  583 = 'S2 583 Row 59 Lost Return Position... Check Ixxx.x Default' | German: 'S2 583 Row 59 Lost Return Position... Check Ixxx.x German' | French: 'S2 583 Row 59 Lost Return Position... Check Ixxx.x French'
  584 = 'S2 584 Row 59 Switch Fault... Check Ixxx.x / Ixxx.x Default' | German: 'S2 584 Row 59 Switch Fault... Check Ixxx.x / Ixxx.x German' | French: 'S2 584 Row 59 Switch Fault... Check Ixxx.x / Ixxx.x French'
  585 = 'S2 585 Row 59 Spare Message Default' | German: 'S2 585 Row 59 Spare Message German' | French: 'S2 585 Row 59 Spare Message French'
  586 = 'S2 586 Row 59 Spare Message Default' | German: 'S2 586 Row 59 Spare Message German' | French: 'S2 586 Row 59 Spare Message French'
  587 = 'S2 587 Row 59 Spare Message Default' | German: 'S2 587 Row 59 Spare Message German' | French: 'S2 587 Row 59 Spare Message French'
  588 = 'S2 588 Row 59 Spare Message Default' | German: 'S2 588 Row 59 Spare Message German' | French: 'S2 588 Row 59 Spare Message French'
  589 = 'S2 589 Row 59 Spare Message Default' | German: 'S2 589 Row 59 Spare Message German' | French: 'S2 589 Row 59 Spare Message French'
  590 = 'S2 590 Row 60 Failed To Advance.. Check Qxxx.x Default' | German: 'S2 590 Row 60 Failed To Advance.. Check Qxxx.x German' | French: 'S2 590 Row 60 Failed To Advance.. Check Qxxx.x French'
  591 = 'S2 591 Row 60 Failed To Return.. Check Qxxx.x Default' | German: 'S2 591 Row 60 Failed To Return.. Check Qxxx.x German' | French: 'S2 591 Row 60 Failed To Return.. Check Qxxx.x French'
  592 = 'S2 592 Row 60 Lost Advance Position... Check Ixxx.x Default' | German: 'S2 592 Row 60 Lost Advance Position... Check Ixxx.x German' | French: 'S2 592 Row 60 Lost Advance Position... Check Ixxx.x French'
  593 = 'S2 593 Row 60 Lost Return Position... Check Ixxx.x Default' | German: 'S2 593 Row 60 Lost Return Position... Check Ixxx.x German' | French: 'S2 593 Row 60 Lost Return Position... Check Ixxx.x French'
  594 = 'S2 594 Row 60 Switch Fault... Check Ixxx.x / Ixxx.x Default' | German: 'S2 594 Row 60 Switch Fault... Check Ixxx.x / Ixxx.x German' | French: 'S2 594 Row 60 Switch Fault... Check Ixxx.x / Ixxx.x French'
  595 = 'S2 595 Row 60 Spare Message Default' | German: 'S2 595 Row 60 Spare Message German' | French: 'S2 595 Row 60 Spare Message French'
  596 = 'S2 596 Row 60 Spare Message Default' | German: 'S2 596 Row 60 Spare Message German' | French: 'S2 596 Row 60 Spare Message French'
  597 = 'S2 597 Row 60 Spare Message Default' | German: 'S2 597 Row 60 Spare Message German' | French: 'S2 597 Row 60 Spare Message French'
  598 = 'S2 598 Row 60 Spare Message Default' | German: 'S2 598 Row 60 Spare Message German' | French: 'S2 598 Row 60 Spare Message French'
  599 = 'S2 599 Row 60 Spare Message Default' | German: 'S2 599 Row 60 Spare Message German' | French: 'S2 599 Row 60 Spare Message French'
  600 = 'S2 600 Row 61 Failed To Advance.. Check Qxxx.x Default' | German: 'S2 600 Row 61 Failed To Advance.. Check Qxxx.x German' | French: 'S2 600 Row 61 Failed To Advance.. Check Qxxx.x French'
  601 = 'S2 601 Row 61 Failed To Return.. Check Qxxx.x Default' | German: 'S2 601 Row 61 Failed To Return.. Check Qxxx.x German' | French: 'S2 601 Row 61 Failed To Return.. Check Qxxx.x French'
  602 = 'S2 602 Row 61 Lost Advance Position... Check Ixxx.x Default' | German: 'S2 602 Row 61 Lost Advance Position... Check Ixxx.x German' | French: 'S2 602 Row 61 Lost Advance Position... Check Ixxx.x French'
  603 = 'S2 603 Row 61 Lost Return Position... Check Ixxx.x Default' | German: 'S2 603 Row 61 Lost Return Position... Check Ixxx.x German' | French: 'S2 603 Row 61 Lost Return Position... Check Ixxx.x French'
  604 = 'S2 604 Row 61 Switch Fault... Check Ixxx.x / Ixxx.x Default' | German: 'S2 604 Row 61 Switch Fault... Check Ixxx.x / Ixxx.x German' | French: 'S2 604 Row 61 Switch Fault... Check Ixxx.x / Ixxx.x French'
  605 = 'S2 605 Row 61 Spare Message Default' | German: 'S2 605 Row 61 Spare Message German' | French: 'S2 605 Row 61 Spare Message French'
  606 = 'S2 606 Row 61 Spare Message Default' | German: 'S2 606 Row 61 Spare Message German' | French: 'S2 606 Row 61 Spare Message French'
  607 = 'S2 607 Row 61 Spare Message Default' | German: 'S2 607 Row 61 Spare Message German' | French: 'S2 607 Row 61 Spare Message French'
  608 = 'S2 608 Row 61 Spare Message Default' | German: 'S2 608 Row 61 Spare Message German' | French: 'S2 608 Row 61 Spare Message French'
  609 = 'S2 609 Row 61 Spare Message Default' | German: 'S2 609 Row 61 Spare Message German' | French: 'S2 609 Row 61 Spare Message French'
  610 = 'S2 610 Row 62 Failed To Advance.. Check Qxxx.x Default' | German: 'S2 610 Row 62 Failed To Advance.. Check Qxxx.x German' | French: 'S2 610 Row 62 Failed To Advance.. Check Qxxx.x French'
  611 = 'S2 611 Row 62 Failed To Return.. Check Qxxx.x Default' | German: 'S2 611 Row 62 Failed To Return.. Check Qxxx.x German' | French: 'S2 611 Row 62 Failed To Return.. Check Qxxx.x French'
  612 = 'S2 612 Row 62 Lost Advance Position... Check Ixxx.x Default' | German: 'S2 612 Row 62 Lost Advance Position... Check Ixxx.x German' | French: 'S2 612 Row 62 Lost Advance Position... Check Ixxx.x French'
  613 = 'S2 613 Row 62 Lost Return Position... Check Ixxx.x Default' | German: 'S2 613 Row 62 Lost Return Position... Check Ixxx.x German' | French: 'S2 613 Row 62 Lost Return Position... Check Ixxx.x French'
  614 = 'S2 614 Row 62 Switch Fault... Check Ixxx.x / Ixxx.x Default' | German: 'S2 614 Row 62 Switch Fault... Check Ixxx.x / Ixxx.x German' | French: 'S2 614 Row 62 Switch Fault... Check Ixxx.x / Ixxx.x French'
  615 = 'S2 615 Row 62 Spare Message Default' | German: 'S2 615 Row 62 Spare Message German' | French: 'S2 615 Row 62 Spare Message French'
  616 = 'S2 616 Row 62 Spare Message Default' | German: 'S2 616 Row 62 Spare Message German' | French: 'S2 616 Row 62 Spare Message French'
  617 = 'S2 617 Row 62 Spare Message Default' | German: 'S2 617 Row 62 Spare Message German' | French: 'S2 617 Row 62 Spare Message French'
  618 = 'S2 618 Row 62 Spare Message Default' | German: 'S2 618 Row 62 Spare Message German' | French: 'S2 618 Row 62 Spare Message French'
  619 = 'S2 619 Row 62 Spare Message Default' | German: 'S2 619 Row 62 Spare Message German' | French: 'S2 619 Row 62 Spare Message French'
  620 = 'S2 620 Row 63 Failed To Advance.. Check Qxxx.x Default' | German: 'S2 620 Row 63 Failed To Advance.. Check Qxxx.x German' | French: 'S2 620 Row 63 Failed To Advance.. Check Qxxx.x French'
  621 = 'S2 621 Row 63 Failed To Return.. Check Qxxx.x Default' | German: 'S2 621 Row 63 Failed To Return.. Check Qxxx.x German' | French: 'S2 621 Row 63 Failed To Return.. Check Qxxx.x French'
  622 = 'S2 622 Row 63 Lost Advance Position... Check Ixxx.x Default' | German: 'S2 622 Row 63 Lost Advance Position... Check Ixxx.x German' | French: 'S2 622 Row 63 Lost Advance Position... Check Ixxx.x French'
  623 = 'S2 623 Row 63 Lost Return Position... Check Ixxx.x Default' | German: 'S2 623 Row 63 Lost Return Position... Check Ixxx.x German' | French: 'S2 623 Row 63 Lost Return Position... Check Ixxx.x French'
  624 = 'S2 624 Row 63 Switch Fault... Check Ixxx.x / Ixxx.x Default' | German: 'S2 624 Row 63 Switch Fault... Check Ixxx.x / Ixxx.x German' | French: 'S2 624 Row 63 Switch Fault... Check Ixxx.x / Ixxx.x French'
  625 = 'S2 625 Row 63 Spare Message Default' | German: 'S2 625 Row 63 Spare Message German' | French: 'S2 625 Row 63 Spare Message French'
  626 = 'S2 626 Row 63 Spare Message Default' | German: 'S2 626 Row 63 Spare Message German' | French: 'S2 626 Row 63 Spare Message French'
  627 = 'S2 627 Row 63 Spare Message Default' | German: 'S2 627 Row 63 Spare Message German' | French: 'S2 627 Row 63 Spare Message French'
  628 = 'S2 628 Row 63 Spare Message Default' | German: 'S2 628 Row 63 Spare Message German' | French: 'S2 628 Row 63 Spare Message French'
  629 = 'S2 629 Row 63 Spare Message Default' | German: 'S2 629 Row 63 Spare Message German' | French: 'S2 629 Row 63 Spare Message French'
  630 = 'S2 630 Row 64 Failed To Advance.. Check Qxxx.x Default' | German: 'S2 630 Row 64 Failed To Advance.. Check Qxxx.x German' | French: 'S2 630 Row 64 Failed To Advance.. Check Qxxx.x French'
  631 = 'S2 631 Row 64 Failed To Return.. Check Qxxx.x Default' | German: 'S2 631 Row 64 Failed To Return.. Check Qxxx.x German' | French: 'S2 631 Row 64 Failed To Return.. Check Qxxx.x French'
  632 = 'S2 632 Row 64 Lost Advance Position... Check Ixxx.x Default' | German: 'S2 632 Row 64 Lost Advance Position... Check Ixxx.x German' | French: 'S2 632 Row 64 Lost Advance Position... Check Ixxx.x French'
  633 = 'S2 633 Row 64 Lost Return Position... Check Ixxx.x Default' | German: 'S2 633 Row 64 Lost Return Position... Check Ixxx.x German' | French: 'S2 633 Row 64 Lost Return Position... Check Ixxx.x French'
  634 = 'S2 634 Row 64 Switch Fault... Check Ixxx.x / Ixxx.x Default' | German: 'S2 634 Row 64 Switch Fault... Check Ixxx.x / Ixxx.x German' | French: 'S2 634 Row 64 Switch Fault... Check Ixxx.x / Ixxx.x French'
  635 = 'S2 635 Row 64 Spare Message Default' | German: 'S2 635 Row 64 Spare Message German' | French: 'S2 635 Row 64 Spare Message French'
  636 = 'S2 636 Row 64 Spare Message Default' | German: 'S2 636 Row 64 Spare Message German' | French: 'S2 636 Row 64 Spare Message French'
  637 = 'S2 637 Row 64 Spare Message Default' | German: 'S2 637 Row 64 Spare Message German' | French: 'S2 637 Row 64 Spare Message French'
  638 = 'S2 638 Row 64 Spare Message Default' | German: 'S2 638 Row 64 Spare Message German' | French: 'S2 638 Row 64 Spare Message French'
  639 = 'S2 639 Row 64 Spare Message Default' | German: 'S2 639 Row 64 Spare Message German' | French: 'S2 639 Row 64 Spare Message French'
  640 = 'S2 640 Row 65 Failed To Advance.. Check Qxxx.x Default' | German: 'S2 640 Row 65 Failed To Advance.. Check Qxxx.x German' | French: 'S2 640 Row 65 Failed To Advance.. Check Qxxx.x French'
  641 = 'S2 641 Row 65 Failed To Return.. Check Qxxx.x Default' | German: 'S2 641 Row 65 Failed To Return.. Check Qxxx.x German' | French: 'S2 641 Row 65 Failed To Return.. Check Qxxx.x French'
  642 = 'S2 642 Row 65 Lost Advance Position... Check Ixxx.x Default' | German: 'S2 642 Row 65 Lost Advance Position... Check Ixxx.x German' | French: 'S2 642 Row 65 Lost Advance Position... Check Ixxx.x French'
  643 = 'S2 643 Row 65 Lost Return Position... Check Ixxx.x Default' | German: 'S2 643 Row 65 Lost Return Position... Check Ixxx.x German' | French: 'S2 643 Row 65 Lost Return Position... Check Ixxx.x French'
  644 = 'S2 644 Row 65 Switch Fault... Check Ixxx.x / Ixxx.x Default' | German: 'S2 644 Row 65 Switch Fault... Check Ixxx.x / Ixxx.x German' | French: 'S2 644 Row 65 Switch Fault... Check Ixxx.x / Ixxx.x French'
  645 = 'S2 645 Row 65 Spare Message Default' | German: 'S2 645 Row 65 Spare Message German' | French: 'S2 645 Row 65 Spare Message French'
  646 = 'S2 646 Row 65 Spare Message Default' | German: 'S2 646 Row 65 Spare Message German' | French: 'S2 646 Row 65 Spare Message French'
  647 = 'S2 647 Row 65 Spare Message Default' | German: 'S2 647 Row 65 Spare Message German' | French: 'S2 647 Row 65 Spare Message French'
  648 = 'S2 648 Row 65 Spare Message Default' | German: 'S2 648 Row 65 Spare Message German' | French: 'S2 648 Row 65 Spare Message French'
  649 = 'S2 649 Row 65 Spare Message Default' | German: 'S2 649 Row 65 Spare Message German' | French: 'S2 649 Row 65 Spare Message French'
  650 = 'S2 650 Row 66 Failed To Advance.. Check Qxxx.x Default' | German: 'S2 650 Row 66 Failed To Advance.. Check Qxxx.x German' | French: 'S2 650 Row 66 Failed To Advance.. Check Qxxx.x French'
  651 = 'S2 651 Row 66 Failed To Return.. Check Qxxx.x Default' | German: 'S2 651 Row 66 Failed To Return.. Check Qxxx.x German' | French: 'S2 651 Row 66 Failed To Return.. Check Qxxx.x French'
  652 = 'S2 652 Row 66 Lost Advance Position... Check Ixxx.x Default' | German: 'S2 652 Row 66 Lost Advance Position... Check Ixxx.x German' | French: 'S2 652 Row 66 Lost Advance Position... Check Ixxx.x French'
  653 = 'S2 653 Row 66 Lost Return Position... Check Ixxx.x Default' | German: 'S2 653 Row 66 Lost Return Position... Check Ixxx.x German' | French: 'S2 653 Row 66 Lost Return Position... Check Ixxx.x French'
  654 = 'S2 654 Row 66 Switch Fault... Check Ixxx.x / Ixxx.x Default' | German: 'S2 654 Row 66 Switch Fault... Check Ixxx.x / Ixxx.x German' | French: 'S2 654 Row 66 Switch Fault... Check Ixxx.x / Ixxx.x French'
  655 = 'S2 655 Row 66 Spare Message Default' | German: 'S2 655 Row 66 Spare Message German' | French: 'S2 655 Row 66 Spare Message French'
  656 = 'S2 656 Row 66 Spare Message Default' | German: 'S2 656 Row 66 Spare Message German' | French: 'S2 656 Row 66 Spare Message French'
  657 = 'S2 657 Row 66 Spare Message Default' | German: 'S2 657 Row 66 Spare Message German' | French: 'S2 657 Row 66 Spare Message French'
  658 = 'S2 658 Row 66 Spare Message Default' | German: 'S2 658 Row 66 Spare Message German' | French: 'S2 658 Row 66 Spare Message French'
  659 = 'S2 659 Row 66 Spare Message Default' | German: 'S2 659 Row 66 Spare Message German' | French: 'S2 659 Row 66 Spare Message French'
  660 = 'S2 660 Row 67 Failed To Advance.. Check Qxxx.x Default' | German: 'S2 660 Row 67 Failed To Advance.. Check Qxxx.x German' | French: 'S2 660 Row 67 Failed To Advance.. Check Qxxx.x French'
  661 = 'S2 661 Row 67 Failed To Return.. Check Qxxx.x Default' | German: 'S2 661 Row 67 Failed To Return.. Check Qxxx.x German' | French: 'S2 661 Row 67 Failed To Return.. Check Qxxx.x French'
  662 = 'S2 662 Row 67 Lost Advance Position... Check Ixxx.x Default' | German: 'S2 662 Row 67 Lost Advance Position... Check Ixxx.x German' | French: 'S2 662 Row 67 Lost Advance Position... Check Ixxx.x French'
  663 = 'S2 663 Row 67 Lost Return Position... Check Ixxx.x Default' | German: 'S2 663 Row 67 Lost Return Position... Check Ixxx.x German' | French: 'S2 663 Row 67 Lost Return Position... Check Ixxx.x French'
  664 = 'S2 664 Row 67 Switch Fault... Check Ixxx.x / Ixxx.x Default' | German: 'S2 664 Row 67 Switch Fault... Check Ixxx.x / Ixxx.x German' | French: 'S2 664 Row 67 Switch Fault... Check Ixxx.x / Ixxx.x French'
  665 = 'S2 665 Row 67 Spare Message Default' | German: 'S2 665 Row 67 Spare Message German' | French: 'S2 665 Row 67 Spare Message French'
  666 = 'S2 666 Row 67 Spare Message Default' | German: 'S2 666 Row 67 Spare Message German' | French: 'S2 666 Row 67 Spare Message French'
  667 = 'S2 667 Row 67 Spare Message Default' | German: 'S2 667 Row 67 Spare Message German' | French: 'S2 667 Row 67 Spare Message French'
  668 = 'S2 668 Row 67 Spare Message Default' | German: 'S2 668 Row 67 Spare Message German' | French: 'S2 668 Row 67 Spare Message French'
  669 = 'S2 669 Row 67 Spare Message Default' | German: 'S2 669 Row 67 Spare Message German' | French: 'S2 669 Row 67 Spare Message French'
  670 = 'S2 670 Row 68 Failed To Advance.. Check Qxxx.x Default' | German: 'S2 670 Row 68 Failed To Advance.. Check Qxxx.x German' | French: 'S2 670 Row 68 Failed To Advance.. Check Qxxx.x French'
  671 = 'S2 671 Row 68 Failed To Return.. Check Qxxx.x Default' | German: 'S2 671 Row 68 Failed To Return.. Check Qxxx.x German' | French: 'S2 671 Row 68 Failed To Return.. Check Qxxx.x French'
  672 = 'S2 672 Row 68 Lost Advance Position... Check Ixxx.x Default' | German: 'S2 672 Row 68 Lost Advance Position... Check Ixxx.x German' | French: 'S2 672 Row 68 Lost Advance Position... Check Ixxx.x French'
  673 = 'S2 673 Row 68 Lost Return Position... Check Ixxx.x Default' | German: 'S2 673 Row 68 Lost Return Position... Check Ixxx.x German' | French: 'S2 673 Row 68 Lost Return Position... Check Ixxx.x French'
  674 = 'S2 674 Row 68 Switch Fault... Check Ixxx.x / Ixxx.x Default' | German: 'S2 674 Row 68 Switch Fault... Check Ixxx.x / Ixxx.x German' | French: 'S2 674 Row 68 Switch Fault... Check Ixxx.x / Ixxx.x French'
  675 = 'S2 675 Row 68 Spare Message Default' | German: 'S2 675 Row 68 Spare Message German' | French: 'S2 675 Row 68 Spare Message French'
  676 = 'S2 676 Row 68 Spare Message Default' | German: 'S2 676 Row 68 Spare Message German' | French: 'S2 676 Row 68 Spare Message French'
  677 = 'S2 677 Row 68 Spare Message Default' | German: 'S2 677 Row 68 Spare Message German' | French: 'S2 677 Row 68 Spare Message French'
  678 = 'S2 678 Row 68 Spare Message Default' | German: 'S2 678 Row 68 Spare Message German' | French: 'S2 678 Row 68 Spare Message French'
  679 = 'S2 679 Row 68 Spare Message Default' | German: 'S2 679 Row 68 Spare Message German' | French: 'S2 679 Row 68 Spare Message French'
  680 = 'S2 680 Row 69 Failed To Advance.. Check Qxxx.x Default' | German: 'S2 680 Row 69 Failed To Advance.. Check Qxxx.x German' | French: 'S2 680 Row 69 Failed To Advance.. Check Qxxx.x French'
  681 = 'S2 681 Row 69 Failed To Return.. Check Qxxx.x Default' | German: 'S2 681 Row 69 Failed To Return.. Check Qxxx.x German' | French: 'S2 681 Row 69 Failed To Return.. Check Qxxx.x French'
  682 = 'S2 682 Row 69 Lost Advance Position... Check Ixxx.x Default' | German: 'S2 682 Row 69 Lost Advance Position... Check Ixxx.x German' | French: 'S2 682 Row 69 Lost Advance Position... Check Ixxx.x French'
  683 = 'S2 683 Row 69 Lost Return Position... Check Ixxx.x Default' | German: 'S2 683 Row 69 Lost Return Position... Check Ixxx.x German' | French: 'S2 683 Row 69 Lost Return Position... Check Ixxx.x French'
  684 = 'S2 684 Row 69 Switch Fault... Check Ixxx.x / Ixxx.x Default' | German: 'S2 684 Row 69 Switch Fault... Check Ixxx.x / Ixxx.x German' | French: 'S2 684 Row 69 Switch Fault... Check Ixxx.x / Ixxx.x French'
  685 = 'S2 685 Row 69 Spare Message Default' | German: 'S2 685 Row 69 Spare Message German' | French: 'S2 685 Row 69 Spare Message French'
  686 = 'S2 686 Row 69 Spare Message Default' | German: 'S2 686 Row 69 Spare Message German' | French: 'S2 686 Row 69 Spare Message French'
  687 = 'S2 687 Row 69 Spare Message Default' | German: 'S2 687 Row 69 Spare Message German' | French: 'S2 687 Row 69 Spare Message French'
  688 = 'S2 688 Row 69 Spare Message Default' | German: 'S2 688 Row 69 Spare Message German' | French: 'S2 688 Row 69 Spare Message French'
  689 = 'S2 689 Row 69 Spare Message Default' | German: 'S2 689 Row 69 Spare Message German' | French: 'S2 689 Row 69 Spare Message French'
  690 = 'S2 690 Row 70 Failed To Advance.. Check Qxxx.x Default' | German: 'S2 690 Row 70 Failed To Advance.. Check Qxxx.x German' | French: 'S2 690 Row 70 Failed To Advance.. Check Qxxx.x French'
  691 = 'S2 691 Row 70 Failed To Return.. Check Qxxx.x Default' | German: 'S2 691 Row 70 Failed To Return.. Check Qxxx.x German' | French: 'S2 691 Row 70 Failed To Return.. Check Qxxx.x French'
  692 = 'S2 692 Row 70 Lost Advance Position... Check Ixxx.x Default' | German: 'S2 692 Row 70 Lost Advance Position... Check Ixxx.x German' | French: 'S2 692 Row 70 Lost Advance Position... Check Ixxx.x French'
  693 = 'S2 693 Row 70 Lost Return Position... Check Ixxx.x Default' | German: 'S2 693 Row 70 Lost Return Position... Check Ixxx.x German' | French: 'S2 693 Row 70 Lost Return Position... Check Ixxx.x French'
  694 = 'S2 694 Row 70 Switch Fault... Check Ixxx.x / Ixxx.x Default' | German: 'S2 694 Row 70 Switch Fault... Check Ixxx.x / Ixxx.x German' | French: 'S2 694 Row 70 Switch Fault... Check Ixxx.x / Ixxx.x French'
  695 = 'S2 695 Row 70 Spare Message Default' | German: 'S2 695 Row 70 Spare Message German' | French: 'S2 695 Row 70 Spare Message French'
  696 = 'S2 696 Row 70 Spare Message Default' | German: 'S2 696 Row 70 Spare Message German' | French: 'S2 696 Row 70 Spare Message French'
  697 = 'S2 697 Row 70 Spare Message Default' | German: 'S2 697 Row 70 Spare Message German' | French: 'S2 697 Row 70 Spare Message French'
  698 = 'S2 698 Row 70 Spare Message Default' | German: 'S2 698 Row 70 Spare Message German' | French: 'S2 698 Row 70 Spare Message French'
  699 = 'S2 699 Row 70 Spare Message Default' | German: 'S2 699 Row 70 Spare Message German' | French: 'S2 699 Row 70 Spare Message French'
  700 = 'S2 700 Row 71 Failed To Advance.. Check Qxxx.x Default' | German: 'S2 700 Row 71 Failed To Advance.. Check Qxxx.x German' | French: 'S2 700 Row 71 Failed To Advance.. Check Qxxx.x French'
  701 = 'S2 701 Row 71 Failed To Return.. Check Qxxx.x Default' | German: 'S2 701 Row 71 Failed To Return.. Check Qxxx.x German' | French: 'S2 701 Row 71 Failed To Return.. Check Qxxx.x French'
  702 = 'S2 702 Row 71 Lost Advance Position... Check Ixxx.x Default' | German: 'S2 702 Row 71 Lost Advance Position... Check Ixxx.x German' | French: 'S2 702 Row 71 Lost Advance Position... Check Ixxx.x French'
  703 = 'S2 703 Row 71 Lost Return Position... Check Ixxx.x Default' | German: 'S2 703 Row 71 Lost Return Position... Check Ixxx.x German' | French: 'S2 703 Row 71 Lost Return Position... Check Ixxx.x French'
  704 = 'S2 704 Row 71 Switch Fault... Check Ixxx.x / Ixxx.x Default' | German: 'S2 704 Row 71 Switch Fault... Check Ixxx.x / Ixxx.x German' | French: 'S2 704 Row 71 Switch Fault... Check Ixxx.x / Ixxx.x French'
  705 = 'S2 705 Row 71 Spare Message Default' | German: 'S2 705 Row 71 Spare Message German' | French: 'S2 705 Row 71 Spare Message French'
  706 = 'S2 706 Row 71 Spare Message Default' | German: 'S2 706 Row 71 Spare Message German' | French: 'S2 706 Row 71 Spare Message French'
  707 = 'S2 707 Row 71 Spare Message Default' | German: 'S2 707 Row 71 Spare Message German' | French: 'S2 707 Row 71 Spare Message French'
  708 = 'S2 708 Row 71 Spare Message Default' | German: 'S2 708 Row 71 Spare Message German' | French: 'S2 708 Row 71 Spare Message French'
  709 = 'S2 709 Row 71 Spare Message Default' | German: 'S2 709 Row 71 Spare Message German' | French: 'S2 709 Row 71 Spare Message French'
  710 = 'S2 710 Row 72 Failed To Advance.. Check Qxxx.x Default' | German: 'S2 710 Row 72 Failed To Advance.. Check Qxxx.x German' | French: 'S2 710 Row 72 Failed To Advance.. Check Qxxx.x French'
  711 = 'S2 711 Row 72 Failed To Return.. Check Qxxx.x Default' | German: 'S2 711 Row 72 Failed To Return.. Check Qxxx.x German' | French: 'S2 711 Row 72 Failed To Return.. Check Qxxx.x French'
  712 = 'S2 712 Row 72 Lost Advance Position... Check Ixxx.x Default' | German: 'S2 712 Row 72 Lost Advance Position... Check Ixxx.x German' | French: 'S2 712 Row 72 Lost Advance Position... Check Ixxx.x French'
  713 = 'S2 713 Row 72 Lost Return Position... Check Ixxx.x Default' | German: 'S2 713 Row 72 Lost Return Position... Check Ixxx.x German' | French: 'S2 713 Row 72 Lost Return Position... Check Ixxx.x French'
  714 = 'S2 714 Row 72 Switch Fault... Check Ixxx.x / Ixxx.x Default' | German: 'S2 714 Row 72 Switch Fault... Check Ixxx.x / Ixxx.x German' | French: 'S2 714 Row 72 Switch Fault... Check Ixxx.x / Ixxx.x French'
  715 = 'S2 715 Row 72 Spare Message Default' | German: 'S2 715 Row 72 Spare Message German' | French: 'S2 715 Row 72 Spare Message French'
  716 = 'S2 716 Row 72 Spare Message Default' | German: 'S2 716 Row 72 Spare Message German' | French: 'S2 716 Row 72 Spare Message French'
  717 = 'S2 717 Row 72 Spare Message Default' | German: 'S2 717 Row 72 Spare Message German' | French: 'S2 717 Row 72 Spare Message French'
  718 = 'S2 718 Row 72 Spare Message Default' | German: 'S2 718 Row 72 Spare Message German' | French: 'S2 718 Row 72 Spare Message French'
  719 = 'S2 719 Row 72 Spare Message Default' | German: 'S2 719 Row 72 Spare Message German' | French: 'S2 719 Row 72 Spare Message French'
  720 = 'S2 720 Row 73 Failed To Advance.. Check Qxxx.x Default' | German: 'S2 720 Row 73 Failed To Advance.. Check Qxxx.x German' | French: 'S2 720 Row 73 Failed To Advance.. Check Qxxx.x French'
  721 = 'S2 721 Row 73 Failed To Return.. Check Qxxx.x Default' | German: 'S2 721 Row 73 Failed To Return.. Check Qxxx.x German' | French: 'S2 721 Row 73 Failed To Return.. Check Qxxx.x French'
  722 = 'S2 722 Row 73 Lost Advance Position... Check Ixxx.x Default' | German: 'S2 722 Row 73 Lost Advance Position... Check Ixxx.x German' | French: 'S2 722 Row 73 Lost Advance Position... Check Ixxx.x French'
  723 = 'S2 723 Row 73 Lost Return Position... Check Ixxx.x Default' | German: 'S2 723 Row 73 Lost Return Position... Check Ixxx.x German' | French: 'S2 723 Row 73 Lost Return Position... Check Ixxx.x French'
  724 = 'S2 724 Row 73 Switch Fault... Check Ixxx.x / Ixxx.x Default' | German: 'S2 724 Row 73 Switch Fault... Check Ixxx.x / Ixxx.x German' | French: 'S2 724 Row 73 Switch Fault... Check Ixxx.x / Ixxx.x French'
  725 = 'S2 725 Row 73 Spare Message Default' | German: 'S2 725 Row 73 Spare Message German' | French: 'S2 725 Row 73 Spare Message French'
  726 = 'S2 726 Row 73 Spare Message Default' | German: 'S2 726 Row 73 Spare Message German' | French: 'S2 726 Row 73 Spare Message French'
  727 = 'S2 727 Row 73 Spare Message Default' | German: 'S2 727 Row 73 Spare Message German' | French: 'S2 727 Row 73 Spare Message French'
  728 = 'S2 728 Row 73 Spare Message Default' | German: 'S2 728 Row 73 Spare Message German' | French: 'S2 728 Row 73 Spare Message French'
  729 = 'S2 729 Row 73 Spare Message Default' | German: 'S2 729 Row 73 Spare Message German' | French: 'S2 729 Row 73 Spare Message French'
  730 = 'S2 730 Row 74 Failed To Advance.. Check Qxxx.x Default' | German: 'S2 730 Row 74 Failed To Advance.. Check Qxxx.x German' | French: 'S2 730 Row 74 Failed To Advance.. Check Qxxx.x French'
  731 = 'S2 731 Row 74 Failed To Return.. Check Qxxx.x Default' | German: 'S2 731 Row 74 Failed To Return.. Check Qxxx.x German' | French: 'S2 731 Row 74 Failed To Return.. Check Qxxx.x French'
  732 = 'S2 732 Row 74 Lost Advance Position... Check Ixxx.x Default' | German: 'S2 732 Row 74 Lost Advance Position... Check Ixxx.x German' | French: 'S2 732 Row 74 Lost Advance Position... Check Ixxx.x French'
  733 = 'S2 733 Row 74 Lost Return Position... Check Ixxx.x Default' | German: 'S2 733 Row 74 Lost Return Position... Check Ixxx.x German' | French: 'S2 733 Row 74 Lost Return Position... Check Ixxx.x French'
  734 = 'S2 734 Row 74 Switch Fault... Check Ixxx.x / Ixxx.x Default' | German: 'S2 734 Row 74 Switch Fault... Check Ixxx.x / Ixxx.x German' | French: 'S2 734 Row 74 Switch Fault... Check Ixxx.x / Ixxx.x French'
  735 = 'S2 735 Row 74 Spare Message Default' | German: 'S2 735 Row 74 Spare Message German' | French: 'S2 735 Row 74 Spare Message French'
  736 = 'S2 736 Row 74 Spare Message Default' | German: 'S2 736 Row 74 Spare Message German' | French: 'S2 736 Row 74 Spare Message French'
  737 = 'S2 737 Row 74 Spare Message Default' | German: 'S2 737 Row 74 Spare Message German' | French: 'S2 737 Row 74 Spare Message French'
  738 = 'S2 738 Row 74 Spare Message Default' | German: 'S2 738 Row 74 Spare Message German' | French: 'S2 738 Row 74 Spare Message French'
  739 = 'S2 739 Row 74 Spare Message Default' | German: 'S2 739 Row 74 Spare Message German' | French: 'S2 739 Row 74 Spare Message French'
  740 = 'S2 740 Row 75 Failed To Advance.. Check Qxxx.x Default' | German: 'S2 740 Row 75 Failed To Advance.. Check Qxxx.x German' | French: 'S2 740 Row 75 Failed To Advance.. Check Qxxx.x French'
  741 = 'S2 741 Row 75 Failed To Return.. Check Qxxx.x Default' | German: 'S2 741 Row 75 Failed To Return.. Check Qxxx.x German' | French: 'S2 741 Row 75 Failed To Return.. Check Qxxx.x French'
  742 = 'S2 742 Row 75 Lost Advance Position... Check Ixxx.x Default' | German: 'S2 742 Row 75 Lost Advance Position... Check Ixxx.x German' | French: 'S2 742 Row 75 Lost Advance Position... Check Ixxx.x French'
  743 = 'S2 743 Row 75 Lost Return Position... Check Ixxx.x Default' | German: 'S2 743 Row 75 Lost Return Position... Check Ixxx.x German' | French: 'S2 743 Row 75 Lost Return Position... Check Ixxx.x French'
  744 = 'S2 744 Row 75 Switch Fault... Check Ixxx.x / Ixxx.x Default' | German: 'S2 744 Row 75 Switch Fault... Check Ixxx.x / Ixxx.x German' | French: 'S2 744 Row 75 Switch Fault... Check Ixxx.x / Ixxx.x French'
  745 = 'S2 745 Row 75 Spare Message Default' | German: 'S2 745 Row 75 Spare Message German' | French: 'S2 745 Row 75 Spare Message French'
  746 = 'S2 746 Row 75 Spare Message Default' | German: 'S2 746 Row 75 Spare Message German' | French: 'S2 746 Row 75 Spare Message French'
  747 = 'S2 747 Row 75 Spare Message Default' | German: 'S2 747 Row 75 Spare Message German' | French: 'S2 747 Row 75 Spare Message French'
  748 = 'S2 748 Row 75 Spare Message Default' | German: 'S2 748 Row 75 Spare Message German' | French: 'S2 748 Row 75 Spare Message French'
  749 = 'S2 749 Row 75 Spare Message Default' | German: 'S2 749 Row 75 Spare Message German' | French: 'S2 749 Row 75 Spare Message French'
  750 = 'S2 750 Row 76 Failed To Advance.. Check Qxxx.x Default' | German: 'S2 750 Row 76 Failed To Advance.. Check Qxxx.x German' | French: 'S2 750 Row 76 Failed To Advance.. Check Qxxx.x French'
  751 = 'S2 751 Row 76 Failed To Return.. Check Qxxx.x Default' | German: 'S2 751 Row 76 Failed To Return.. Check Qxxx.x German' | French: 'S2 751 Row 76 Failed To Return.. Check Qxxx.x French'
  752 = 'S2 752 Row 76 Lost Advance Position... Check Ixxx.x Default' | German: 'S2 752 Row 76 Lost Advance Position... Check Ixxx.x German' | French: 'S2 752 Row 76 Lost Advance Position... Check Ixxx.x French'
  753 = 'S2 753 Row 76 Lost Return Position... Check Ixxx.x Default' | German: 'S2 753 Row 76 Lost Return Position... Check Ixxx.x German' | French: 'S2 753 Row 76 Lost Return Position... Check Ixxx.x French'
  754 = 'S2 754 Row 76 Switch Fault... Check Ixxx.x / Ixxx.x Default' | German: 'S2 754 Row 76 Switch Fault... Check Ixxx.x / Ixxx.x German' | French: 'S2 754 Row 76 Switch Fault... Check Ixxx.x / Ixxx.x French'
  755 = 'S2 755 Row 76 Spare Message Default' | German: 'S2 755 Row 76 Spare Message German' | French: 'S2 755 Row 76 Spare Message French'
  756 = 'S2 756 Row 76 Spare Message Default' | German: 'S2 756 Row 76 Spare Message German' | French: 'S2 756 Row 76 Spare Message French'
  757 = 'S2 757 Row 76 Spare Message Default' | German: 'S2 757 Row 76 Spare Message German' | French: 'S2 757 Row 76 Spare Message French'
  758 = 'S2 758 Row 76 Spare Message Default' | German: 'S2 758 Row 76 Spare Message German' | French: 'S2 758 Row 76 Spare Message French'
  759 = 'S2 759 Row 76 Spare Message Default' | German: 'S2 759 Row 76 Spare Message German' | French: 'S2 759 Row 76 Spare Message French'
  760 = 'S2 760 Row 77 Failed To Advance.. Check Qxxx.x Default' | German: 'S2 760 Row 77 Failed To Advance.. Check Qxxx.x German' | French: 'S2 760 Row 77 Failed To Advance.. Check Qxxx.x French'
  761 = 'S2 761 Row 77 Failed To Return.. Check Qxxx.x Default' | German: 'S2 761 Row 77 Failed To Return.. Check Qxxx.x German' | French: 'S2 761 Row 77 Failed To Return.. Check Qxxx.x French'
  762 = 'S2 762 Row 77 Lost Advance Position... Check Ixxx.x Default' | German: 'S2 762 Row 77 Lost Advance Position... Check Ixxx.x German' | French: 'S2 762 Row 77 Lost Advance Position... Check Ixxx.x French'
  763 = 'S2 763 Row 77 Lost Return Position... Check Ixxx.x Default' | German: 'S2 763 Row 77 Lost Return Position... Check Ixxx.x German' | French: 'S2 763 Row 77 Lost Return Position... Check Ixxx.x French'
  764 = 'S2 764 Row 77 Switch Fault... Check Ixxx.x / Ixxx.x Default' | German: 'S2 764 Row 77 Switch Fault... Check Ixxx.x / Ixxx.x German' | French: 'S2 764 Row 77 Switch Fault... Check Ixxx.x / Ixxx.x French'
  765 = 'S2 765 Row 77 Spare Message Default' | German: 'S2 765 Row 77 Spare Message German' | French: 'S2 765 Row 77 Spare Message French'
  766 = 'S2 766 Row 77 Spare Message Default' | German: 'S2 766 Row 77 Spare Message German' | French: 'S2 766 Row 77 Spare Message French'
  767 = 'S2 767 Row 77 Spare Message Default' | German: 'S2 767 Row 77 Spare Message German' | French: 'S2 767 Row 77 Spare Message French'
  768 = 'S2 768 Row 77 Spare Message Default' | German: 'S2 768 Row 77 Spare Message German' | French: 'S2 768 Row 77 Spare Message French'
  769 = 'S2 769 Row 77 Spare Message Default' | German: 'S2 769 Row 77 Spare Message German' | French: 'S2 769 Row 77 Spare Message French'
  770 = 'S2 770 Row 78 Failed To Advance.. Check Qxxx.x Default' | German: 'S2 770 Row 78 Failed To Advance.. Check Qxxx.x German' | French: 'S2 770 Row 78 Failed To Advance.. Check Qxxx.x French'
  771 = 'S2 771 Row 78 Failed To Return.. Check Qxxx.x Default' | German: 'S2 771 Row 78 Failed To Return.. Check Qxxx.x German' | French: 'S2 771 Row 78 Failed To Return.. Check Qxxx.x French'
  772 = 'S2 772 Row 78 Lost Advance Position... Check Ixxx.x Default' | German: 'S2 772 Row 78 Lost Advance Position... Check Ixxx.x German' | French: 'S2 772 Row 78 Lost Advance Position... Check Ixxx.x French'
  773 = 'S2 773 Row 78 Lost Return Position... Check Ixxx.x Default' | German: 'S2 773 Row 78 Lost Return Position... Check Ixxx.x German' | French: 'S2 773 Row 78 Lost Return Position... Check Ixxx.x French'
  774 = 'S2 774 Row 78 Switch Fault... Check Ixxx.x / Ixxx.x Default' | German: 'S2 774 Row 78 Switch Fault... Check Ixxx.x / Ixxx.x German' | French: 'S2 774 Row 78 Switch Fault... Check Ixxx.x / Ixxx.x French'
  775 = 'S2 775 Row 78 Spare Message Default' | German: 'S2 775 Row 78 Spare Message German' | French: 'S2 775 Row 78 Spare Message French'
  776 = 'S2 776 Row 78 Spare Message Default' | German: 'S2 776 Row 78 Spare Message German' | French: 'S2 776 Row 78 Spare Message French'
  777 = 'S2 777 Row 78 Spare Message Default' | German: 'S2 777 Row 78 Spare Message German' | French: 'S2 777 Row 78 Spare Message French'
  778 = 'S2 778 Row 78 Spare Message Default' | German: 'S2 778 Row 78 Spare Message German' | French: 'S2 778 Row 78 Spare Message French'
  779 = 'S2 779 Row 78 Spare Message Default' | German: 'S2 779 Row 78 Spare Message German' | French: 'S2 779 Row 78 Spare Message French'
  780 = 'S2 780 Row 79 Failed To Advance.. Check Qxxx.x Default' | German: 'S2 780 Row 79 Failed To Advance.. Check Qxxx.x German' | French: 'S2 780 Row 79 Failed To Advance.. Check Qxxx.x French'
  781 = 'S2 781 Row 79 Failed To Return.. Check Qxxx.x Default' | German: 'S2 781 Row 79 Failed To Return.. Check Qxxx.x German' | French: 'S2 781 Row 79 Failed To Return.. Check Qxxx.x French'
  782 = 'S2 782 Row 79 Lost Advance Position... Check Ixxx.x Default' | German: 'S2 782 Row 79 Lost Advance Position... Check Ixxx.x German' | French: 'S2 782 Row 79 Lost Advance Position... Check Ixxx.x French'
  783 = 'S2 783 Row 79 Lost Return Position... Check Ixxx.x Default' | German: 'S2 783 Row 79 Lost Return Position... Check Ixxx.x German' | French: 'S2 783 Row 79 Lost Return Position... Check Ixxx.x French'
  784 = 'S2 784 Row 79 Switch Fault... Check Ixxx.x / Ixxx.x Default' | German: 'S2 784 Row 79 Switch Fault... Check Ixxx.x / Ixxx.x German' | French: 'S2 784 Row 79 Switch Fault... Check Ixxx.x / Ixxx.x French'
  785 = 'S2 785 Row 79 Spare Message Default' | German: 'S2 785 Row 79 Spare Message German' | French: 'S2 785 Row 79 Spare Message French'
  786 = 'S2 786 Row 79 Spare Message Default' | German: 'S2 786 Row 79 Spare Message German' | French: 'S2 786 Row 79 Spare Message French'
  787 = 'S2 787 Row 79 Spare Message Default' | German: 'S2 787 Row 79 Spare Message German' | French: 'S2 787 Row 79 Spare Message French'
  788 = 'S2 788 Row 79 Spare Message Default' | German: 'S2 788 Row 79 Spare Message German' | French: 'S2 788 Row 79 Spare Message French'
  789 = 'S2 789 Row 79 Spare Message Default' | German: 'S2 789 Row 79 Spare Message German' | French: 'S2 789 Row 79 Spare Message French'
  790 = 'S2 790 Row 80 Failed To Advance.. Check Qxxx.x Default' | German: 'S2 790 Row 80 Failed To Advance.. Check Qxxx.x German' | French: 'S2 790 Row 80 Failed To Advance.. Check Qxxx.x French'
  791 = 'S2 791 Row 80 Failed To Return.. Check Qxxx.x Default' | German: 'S2 791 Row 80 Failed To Return.. Check Qxxx.x German' | French: 'S2 791 Row 80 Failed To Return.. Check Qxxx.x French'
  792 = 'S2 792 Row 80 Lost Advance Position... Check Ixxx.x Default' | German: 'S2 792 Row 80 Lost Advance Position... Check Ixxx.x German' | French: 'S2 792 Row 80 Lost Advance Position... Check Ixxx.x French'
  793 = 'S2 793 Row 80 Lost Return Position... Check Ixxx.x Default' | German: 'S2 793 Row 80 Lost Return Position... Check Ixxx.x German' | French: 'S2 793 Row 80 Lost Return Position... Check Ixxx.x French'
  794 = 'S2 794 Row 80 Switch Fault... Check Ixxx.x / Ixxx.x Default' | German: 'S2 794 Row 80 Switch Fault... Check Ixxx.x / Ixxx.x German' | French: 'S2 794 Row 80 Switch Fault... Check Ixxx.x / Ixxx.x French'
  795 = 'S2 795 Row 80 Spare Message Default' | German: 'S2 795 Row 80 Spare Message German' | French: 'S2 795 Row 80 Spare Message French'
  796 = 'S2 796 Row 80 Spare Message Default' | German: 'S2 796 Row 80 Spare Message German' | French: 'S2 796 Row 80 Spare Message French'
  797 = 'S2 797 Row 80 Spare Message Default' | German: 'S2 797 Row 80 Spare Message German' | French: 'S2 797 Row 80 Spare Message French'
  798 = 'S2 798 Row 80 Spare Message Default' | German: 'S2 798 Row 80 Spare Message German' | French: 'S2 798 Row 80 Spare Message French'
  799 = 'S2 799 Row 80 Spare Message Default' | German: 'S2 799 Row 80 Spare Message German' | French: 'S2 799 Row 80 Spare Message French'
  800 = 'S2 800 Row 81 Failed To Advance.. Check Qxxx.x Default' | German: 'S2 800 Row 81 Failed To Advance.. Check Qxxx.x German' | French: 'S2 800 Row 81 Failed To Advance.. Check Qxxx.x French'
  801 = 'S2 801 Row 81 Failed To Return.. Check Qxxx.x Default' | German: 'S2 801 Row 81 Failed To Return.. Check Qxxx.x German' | French: 'S2 801 Row 81 Failed To Return.. Check Qxxx.x French'
  802 = 'S2 802 Row 81 Lost Advance Position... Check Ixxx.x Default' | German: 'S2 802 Row 81 Lost Advance Position... Check Ixxx.x German' | French: 'S2 802 Row 81 Lost Advance Position... Check Ixxx.x French'
  803 = 'S2 803 Row 81 Lost Return Position... Check Ixxx.x Default' | German: 'S2 803 Row 81 Lost Return Position... Check Ixxx.x German' | French: 'S2 803 Row 81 Lost Return Position... Check Ixxx.x French'
  804 = 'S2 804 Row 81 Switch Fault... Check Ixxx.x / Ixxx.x Default' | German: 'S2 804 Row 81 Switch Fault... Check Ixxx.x / Ixxx.x German' | French: 'S2 804 Row 81 Switch Fault... Check Ixxx.x / Ixxx.x French'
  805 = 'S2 805 Row 81 Spare Message Default' | German: 'S2 805 Row 81 Spare Message German' | French: 'S2 805 Row 81 Spare Message French'
  806 = 'S2 806 Row 81 Spare Message Default' | German: 'S2 806 Row 81 Spare Message German' | French: 'S2 806 Row 81 Spare Message French'
  807 = 'S2 807 Row 81 Spare Message Default' | German: 'S2 807 Row 81 Spare Message German' | French: 'S2 807 Row 81 Spare Message French'
  808 = 'S2 808 Row 81 Spare Message Default' | German: 'S2 808 Row 81 Spare Message German' | French: 'S2 808 Row 81 Spare Message French'
  809 = 'S2 809 Row 81 Spare Message Default' | German: 'S2 809 Row 81 Spare Message German' | French: 'S2 809 Row 81 Spare Message French'
  810 = 'S2 810 Row 82 Failed To Advance.. Check Qxxx.x Default' | German: 'S2 810 Row 82 Failed To Advance.. Check Qxxx.x German' | French: 'S2 810 Row 82 Failed To Advance.. Check Qxxx.x French'
  811 = 'S2 811 Row 82 Failed To Return.. Check Qxxx.x Default' | German: 'S2 811 Row 82 Failed To Return.. Check Qxxx.x German' | French: 'S2 811 Row 82 Failed To Return.. Check Qxxx.x French'
  812 = 'S2 812 Row 82 Lost Advance Position... Check Ixxx.x Default' | German: 'S2 812 Row 82 Lost Advance Position... Check Ixxx.x German' | French: 'S2 812 Row 82 Lost Advance Position... Check Ixxx.x French'
  813 = 'S2 813 Row 82 Lost Return Position... Check Ixxx.x Default' | German: 'S2 813 Row 82 Lost Return Position... Check Ixxx.x German' | French: 'S2 813 Row 82 Lost Return Position... Check Ixxx.x French'
  814 = 'S2 814 Row 82 Switch Fault... Check Ixxx.x / Ixxx.x Default' | German: 'S2 814 Row 82 Switch Fault... Check Ixxx.x / Ixxx.x German' | French: 'S2 814 Row 82 Switch Fault... Check Ixxx.x / Ixxx.x French'
  815 = 'S2 815 Row 82 Spare Message Default' | German: 'S2 815 Row 82 Spare Message German' | French: 'S2 815 Row 82 Spare Message French'
  816 = 'S2 816 Row 82 Spare Message Default' | German: 'S2 816 Row 82 Spare Message German' | French: 'S2 816 Row 82 Spare Message French'
  817 = 'S2 817 Row 82 Spare Message Default' | German: 'S2 817 Row 82 Spare Message German' | French: 'S2 817 Row 82 Spare Message French'
  818 = 'S2 818 Row 82 Spare Message Default' | German: 'S2 818 Row 82 Spare Message German' | French: 'S2 818 Row 82 Spare Message French'
  819 = 'S2 819 Row 82 Spare Message Default' | German: 'S2 819 Row 82 Spare Message German' | French: 'S2 819 Row 82 Spare Message French'
  820 = 'S2 820 Row 83 Failed To Advance.. Check Qxxx.x Default' | German: 'S2 820 Row 83 Failed To Advance.. Check Qxxx.x German' | French: 'S2 820 Row 83 Failed To Advance.. Check Qxxx.x French'
  821 = 'S2 821 Row 83 Failed To Return.. Check Qxxx.x Default' | German: 'S2 821 Row 83 Failed To Return.. Check Qxxx.x German' | French: 'S2 821 Row 83 Failed To Return.. Check Qxxx.x French'
  822 = 'S2 822 Row 83 Lost Advance Position... Check Ixxx.x Default' | German: 'S2 822 Row 83 Lost Advance Position... Check Ixxx.x German' | French: 'S2 822 Row 83 Lost Advance Position... Check Ixxx.x French'
  823 = 'S2 823 Row 83 Lost Return Position... Check Ixxx.x Default' | German: 'S2 823 Row 83 Lost Return Position... Check Ixxx.x German' | French: 'S2 823 Row 83 Lost Return Position... Check Ixxx.x French'
  824 = 'S2 824 Row 83 Switch Fault... Check Ixxx.x / Ixxx.x Default' | German: 'S2 824 Row 83 Switch Fault... Check Ixxx.x / Ixxx.x German' | French: 'S2 824 Row 83 Switch Fault... Check Ixxx.x / Ixxx.x French'
  825 = 'S2 825 Row 83 Spare Message Default' | German: 'S2 825 Row 83 Spare Message German' | French: 'S2 825 Row 83 Spare Message French'
  826 = 'S2 826 Row 83 Spare Message Default' | German: 'S2 826 Row 83 Spare Message German' | French: 'S2 826 Row 83 Spare Message French'
  827 = 'S2 827 Row 83 Spare Message Default' | German: 'S2 827 Row 83 Spare Message German' | French: 'S2 827 Row 83 Spare Message French'
  828 = 'S2 828 Row 83 Spare Message Default' | German: 'S2 828 Row 83 Spare Message German' | French: 'S2 828 Row 83 Spare Message French'
  829 = 'S2 829 Row 83 Spare Message Default' | German: 'S2 829 Row 83 Spare Message German' | French: 'S2 829 Row 83 Spare Message French'
  830 = 'S2 830 Row 84 Failed To Advance.. Check Qxxx.x Default' | German: 'S2 830 Row 84 Failed To Advance.. Check Qxxx.x German' | French: 'S2 830 Row 84 Failed To Advance.. Check Qxxx.x French'
  831 = 'S2 831 Row 84 Failed To Return.. Check Qxxx.x Default' | German: 'S2 831 Row 84 Failed To Return.. Check Qxxx.x German' | French: 'S2 831 Row 84 Failed To Return.. Check Qxxx.x French'
  832 = 'S2 832 Row 84 Lost Advance Position... Check Ixxx.x Default' | German: 'S2 832 Row 84 Lost Advance Position... Check Ixxx.x German' | French: 'S2 832 Row 84 Lost Advance Position... Check Ixxx.x French'
  833 = 'S2 833 Row 84 Lost Return Position... Check Ixxx.x Default' | German: 'S2 833 Row 84 Lost Return Position... Check Ixxx.x German' | French: 'S2 833 Row 84 Lost Return Position... Check Ixxx.x French'
  834 = 'S2 834 Row 84 Switch Fault... Check Ixxx.x / Ixxx.x Default' | German: 'S2 834 Row 84 Switch Fault... Check Ixxx.x / Ixxx.x German' | French: 'S2 834 Row 84 Switch Fault... Check Ixxx.x / Ixxx.x French'
  835 = 'S2 835 Row 84 Spare Message Default' | German: 'S2 835 Row 84 Spare Message German' | French: 'S2 835 Row 84 Spare Message French'
  836 = 'S2 836 Row 84 Spare Message Default' | German: 'S2 836 Row 84 Spare Message German' | French: 'S2 836 Row 84 Spare Message French'
  837 = 'S2 837 Row 84 Spare Message Default' | German: 'S2 837 Row 84 Spare Message German' | French: 'S2 837 Row 84 Spare Message French'
  838 = 'S2 838 Row 84 Spare Message Default' | German: 'S2 838 Row 84 Spare Message German' | French: 'S2 838 Row 84 Spare Message French'
  839 = 'S2 839 Row 84 Spare Message Default' | German: 'S2 839 Row 84 Spare Message German' | French: 'S2 839 Row 84 Spare Message French'
  840 = 'S2 840 Row 85 Failed To Advance.. Check Qxxx.x Default' | German: 'S2 840 Row 85 Failed To Advance.. Check Qxxx.x German' | French: 'S2 840 Row 85 Failed To Advance.. Check Qxxx.x French'
  841 = 'S2 841 Row 85 Failed To Return.. Check Qxxx.x Default' | German: 'S2 841 Row 85 Failed To Return.. Check Qxxx.x German' | French: 'S2 841 Row 85 Failed To Return.. Check Qxxx.x French'
  842 = 'S2 842 Row 85 Lost Advance Position... Check Ixxx.x Default' | German: 'S2 842 Row 85 Lost Advance Position... Check Ixxx.x German' | French: 'S2 842 Row 85 Lost Advance Position... Check Ixxx.x French'
  843 = 'S2 843 Row 85 Lost Return Position... Check Ixxx.x Default' | German: 'S2 843 Row 85 Lost Return Position... Check Ixxx.x German' | French: 'S2 843 Row 85 Lost Return Position... Check Ixxx.x French'
  844 = 'S2 844 Row 85 Switch Fault... Check Ixxx.x / Ixxx.x Default' | German: 'S2 844 Row 85 Switch Fault... Check Ixxx.x / Ixxx.x German' | French: 'S2 844 Row 85 Switch Fault... Check Ixxx.x / Ixxx.x French'
  845 = 'S2 845 Row 85 Spare Message Default' | German: 'S2 845 Row 85 Spare Message German' | French: 'S2 845 Row 85 Spare Message French'
  846 = 'S2 846 Row 85 Spare Message Default' | German: 'S2 846 Row 85 Spare Message German' | French: 'S2 846 Row 85 Spare Message French'
  847 = 'S2 847 Row 85 Spare Message Default' | German: 'S2 847 Row 85 Spare Message German' | French: 'S2 847 Row 85 Spare Message French'
  848 = 'S2 848 Row 85 Spare Message Default' | German: 'S2 848 Row 85 Spare Message German' | French: 'S2 848 Row 85 Spare Message French'
  849 = 'S2 849 Row 85 Spare Message Default' | German: 'S2 849 Row 85 Spare Message German' | French: 'S2 849 Row 85 Spare Message French'
  850 = 'S2 850 Row 86 Failed To Advance.. Check Qxxx.x Default' | German: 'S2 850 Row 86 Failed To Advance.. Check Qxxx.x German' | French: 'S2 850 Row 86 Failed To Advance.. Check Qxxx.x French'
  851 = 'S2 851 Row 86 Failed To Return.. Check Qxxx.x Default' | German: 'S2 851 Row 86 Failed To Return.. Check Qxxx.x German' | French: 'S2 851 Row 86 Failed To Return.. Check Qxxx.x French'
  852 = 'S2 852 Row 86 Lost Advance Position... Check Ixxx.x Default' | German: 'S2 852 Row 86 Lost Advance Position... Check Ixxx.x German' | French: 'S2 852 Row 86 Lost Advance Position... Check Ixxx.x French'
  853 = 'S2 853 Row 86 Lost Return Position... Check Ixxx.x Default' | German: 'S2 853 Row 86 Lost Return Position... Check Ixxx.x German' | French: 'S2 853 Row 86 Lost Return Position... Check Ixxx.x French'
  854 = 'S2 854 Row 86 Switch Fault... Check Ixxx.x / Ixxx.x Default' | German: 'S2 854 Row 86 Switch Fault... Check Ixxx.x / Ixxx.x German' | French: 'S2 854 Row 86 Switch Fault... Check Ixxx.x / Ixxx.x French'
  855 = 'S2 855 Row 86 Spare Message Default' | German: 'S2 855 Row 86 Spare Message German' | French: 'S2 855 Row 86 Spare Message French'
  856 = 'S2 856 Row 86 Spare Message Default' | German: 'S2 856 Row 86 Spare Message German' | French: 'S2 856 Row 86 Spare Message French'
  857 = 'S2 857 Row 86 Spare Message Default' | German: 'S2 857 Row 86 Spare Message German' | French: 'S2 857 Row 86 Spare Message French'
  858 = 'S2 858 Row 86 Spare Message Default' | German: 'S2 858 Row 86 Spare Message German' | French: 'S2 858 Row 86 Spare Message French'
  859 = 'S2 859 Row 86 Spare Message Default' | German: 'S2 859 Row 86 Spare Message German' | French: 'S2 859 Row 86 Spare Message French'
  860 = 'S2 860 Row 87 Failed To Advance.. Check Qxxx.x Default' | German: 'S2 860 Row 87 Failed To Advance.. Check Qxxx.x German' | French: 'S2 860 Row 87 Failed To Advance.. Check Qxxx.x French'
  861 = 'S2 861 Row 87 Failed To Return.. Check Qxxx.x Default' | German: 'S2 861 Row 87 Failed To Return.. Check Qxxx.x German' | French: 'S2 861 Row 87 Failed To Return.. Check Qxxx.x French'
  862 = 'S2 862 Row 87 Lost Advance Position... Check Ixxx.x Default' | German: 'S2 862 Row 87 Lost Advance Position... Check Ixxx.x German' | French: 'S2 862 Row 87 Lost Advance Position... Check Ixxx.x French'
  863 = 'S2 863 Row 87 Lost Return Position... Check Ixxx.x Default' | German: 'S2 863 Row 87 Lost Return Position... Check Ixxx.x German' | French: 'S2 863 Row 87 Lost Return Position... Check Ixxx.x French'
  864 = 'S2 864 Row 87 Switch Fault... Check Ixxx.x / Ixxx.x Default' | German: 'S2 864 Row 87 Switch Fault... Check Ixxx.x / Ixxx.x German' | French: 'S2 864 Row 87 Switch Fault... Check Ixxx.x / Ixxx.x French'
  865 = 'S2 865 Row 87 Spare Message Default' | German: 'S2 865 Row 87 Spare Message German' | French: 'S2 865 Row 87 Spare Message French'
  866 = 'S2 866 Row 87 Spare Message Default' | German: 'S2 866 Row 87 Spare Message German' | French: 'S2 866 Row 87 Spare Message French'
  867 = 'S2 867 Row 87 Spare Message Default' | German: 'S2 867 Row 87 Spare Message German' | French: 'S2 867 Row 87 Spare Message French'
  868 = 'S2 868 Row 87 Spare Message Default' | German: 'S2 868 Row 87 Spare Message German' | French: 'S2 868 Row 87 Spare Message French'
  869 = 'S2 869 Row 87 Spare Message Default' | German: 'S2 869 Row 87 Spare Message German' | French: 'S2 869 Row 87 Spare Message French'
  870 = 'S2 870 Row 88 Failed To Advance.. Check Qxxx.x Default' | German: 'S2 870 Row 88 Failed To Advance.. Check Qxxx.x German' | French: 'S2 870 Row 88 Failed To Advance.. Check Qxxx.x French'
  871 = 'S2 871 Row 88 Failed To Return.. Check Qxxx.x Default' | German: 'S2 871 Row 88 Failed To Return.. Check Qxxx.x German' | French: 'S2 871 Row 88 Failed To Return.. Check Qxxx.x French'
  872 = 'S2 872 Row 88 Lost Advance Position... Check Ixxx.x Default' | German: 'S2 872 Row 88 Lost Advance Position... Check Ixxx.x German' | French: 'S2 872 Row 88 Lost Advance Position... Check Ixxx.x French'
  873 = 'S2 873 Row 88 Lost Return Position... Check Ixxx.x Default' | German: 'S2 873 Row 88 Lost Return Position... Check Ixxx.x German' | French: 'S2 873 Row 88 Lost Return Position... Check Ixxx.x French'
  874 = 'S2 874 Row 88 Switch Fault... Check Ixxx.x / Ixxx.x Default' | German: 'S2 874 Row 88 Switch Fault... Check Ixxx.x / Ixxx.x German' | French: 'S2 874 Row 88 Switch Fault... Check Ixxx.x / Ixxx.x French'
  875 = 'S2 875 Row 88 Spare Message Default' | German: 'S2 875 Row 88 Spare Message German' | French: 'S2 875 Row 88 Spare Message French'
  876 = 'S2 876 Row 88 Spare Message Default' | German: 'S2 876 Row 88 Spare Message German' | French: 'S2 876 Row 88 Spare Message French'
  877 = 'S2 877 Row 88 Spare Message Default' | German: 'S2 877 Row 88 Spare Message German' | French: 'S2 877 Row 88 Spare Message French'
  878 = 'S2 878 Row 88 Spare Message Default' | German: 'S2 878 Row 88 Spare Message German' | French: 'S2 878 Row 88 Spare Message French'
  879 = 'S2 879 Row 88 Spare Message Default' | German: 'S2 879 Row 88 Spare Message German' | French: 'S2 879 Row 88 Spare Message French'
  880 = 'S2 880 Row 89 Failed To Advance.. Check Qxxx.x Default' | German: 'S2 880 Row 89 Failed To Advance.. Check Qxxx.x German' | French: 'S2 880 Row 89 Failed To Advance.. Check Qxxx.x French'
  881 = 'S2 881 Row 89 Failed To Return.. Check Qxxx.x Default' | German: 'S2 881 Row 89 Failed To Return.. Check Qxxx.x German' | French: 'S2 881 Row 89 Failed To Return.. Check Qxxx.x French'
  882 = 'S2 882 Row 89 Lost Advance Position... Check Ixxx.x Default' | German: 'S2 882 Row 89 Lost Advance Position... Check Ixxx.x German' | French: 'S2 882 Row 89 Lost Advance Position... Check Ixxx.x French'
  883 = 'S2 883 Row 89 Lost Return Position... Check Ixxx.x Default' | German: 'S2 883 Row 89 Lost Return Position... Check Ixxx.x German' | French: 'S2 883 Row 89 Lost Return Position... Check Ixxx.x French'
  884 = 'S2 884 Row 89 Switch Fault... Check Ixxx.x / Ixxx.x Default' | German: 'S2 884 Row 89 Switch Fault... Check Ixxx.x / Ixxx.x German' | French: 'S2 884 Row 89 Switch Fault... Check Ixxx.x / Ixxx.x French'
  885 = 'S2 885 Row 89 Spare Message Default' | German: 'S2 885 Row 89 Spare Message German' | French: 'S2 885 Row 89 Spare Message French'
  886 = 'S2 886 Row 89 Spare Message Default' | German: 'S2 886 Row 89 Spare Message German' | French: 'S2 886 Row 89 Spare Message French'
  887 = 'S2 887 Row 89 Spare Message Default' | German: 'S2 887 Row 89 Spare Message German' | French: 'S2 887 Row 89 Spare Message French'
  888 = 'S2 888 Row 89 Spare Message Default' | German: 'S2 888 Row 89 Spare Message German' | French: 'S2 888 Row 89 Spare Message French'
  889 = 'S2 889 Row 89 Spare Message Default' | German: 'S2 889 Row 89 Spare Message German' | French: 'S2 889 Row 89 Spare Message French'
  890 = 'S2 890 Row 90 Failed To Advance.. Check Qxxx.x Default' | German: 'S2 890 Row 90 Failed To Advance.. Check Qxxx.x German' | French: 'S2 890 Row 90 Failed To Advance.. Check Qxxx.x French'
  891 = 'S2 891 Row 90 Failed To Return.. Check Qxxx.x Default' | German: 'S2 891 Row 90 Failed To Return.. Check Qxxx.x German' | French: 'S2 891 Row 90 Failed To Return.. Check Qxxx.x French'
  892 = 'S2 892 Row 90 Lost Advance Position... Check Ixxx.x Default' | German: 'S2 892 Row 90 Lost Advance Position... Check Ixxx.x German' | French: 'S2 892 Row 90 Lost Advance Position... Check Ixxx.x French'
  893 = 'S2 893 Row 90 Lost Return Position... Check Ixxx.x Default' | German: 'S2 893 Row 90 Lost Return Position... Check Ixxx.x German' | French: 'S2 893 Row 90 Lost Return Position... Check Ixxx.x French'
  894 = 'S2 894 Row 90 Switch Fault... Check Ixxx.x / Ixxx.x Default' | German: 'S2 894 Row 90 Switch Fault... Check Ixxx.x / Ixxx.x German' | French: 'S2 894 Row 90 Switch Fault... Check Ixxx.x / Ixxx.x French'
  895 = 'S2 895 Row 90 Spare Message Default' | German: 'S2 895 Row 90 Spare Message German' | French: 'S2 895 Row 90 Spare Message French'
  896 = 'S2 896 Row 90 Spare Message Default' | German: 'S2 896 Row 90 Spare Message German' | French: 'S2 896 Row 90 Spare Message French'
  897 = 'S2 897 Row 90 Spare Message Default' | German: 'S2 897 Row 90 Spare Message German' | French: 'S2 897 Row 90 Spare Message French'
  898 = 'S2 898 Row 90 Spare Message Default' | German: 'S2 898 Row 90 Spare Message German' | French: 'S2 898 Row 90 Spare Message French'
  899 = 'S2 899 Row 90 Spare Message Default' | German: 'S2 899 Row 90 Spare Message German' | French: 'S2 899 Row 90 Spare Message French'
  900 = 'S2 900 Row 91 Failed To Advance.. Check Qxxx.x Default' | German: 'S2 900 Row 91 Failed To Advance.. Check Qxxx.x German' | French: 'S2 900 Row 91 Failed To Advance.. Check Qxxx.x French'
  901 = 'S2 901 Row 91 Failed To Return.. Check Qxxx.x Default' | German: 'S2 901 Row 91 Failed To Return.. Check Qxxx.x German' | French: 'S2 901 Row 91 Failed To Return.. Check Qxxx.x French'
  902 = 'S2 902 Row 91 Lost Advance Position... Check Ixxx.x Default' | German: 'S2 902 Row 91 Lost Advance Position... Check Ixxx.x German' | French: 'S2 902 Row 91 Lost Advance Position... Check Ixxx.x French'
  903 = 'S2 903 Row 91 Lost Return Position... Check Ixxx.x Default' | German: 'S2 903 Row 91 Lost Return Position... Check Ixxx.x German' | French: 'S2 903 Row 91 Lost Return Position... Check Ixxx.x French'
  904 = 'S2 904 Row 91 Switch Fault... Check Ixxx.x / Ixxx.x Default' | German: 'S2 904 Row 91 Switch Fault... Check Ixxx.x / Ixxx.x German' | French: 'S2 904 Row 91 Switch Fault... Check Ixxx.x / Ixxx.x French'
  905 = 'S2 905 Row 91 Spare Message Default' | German: 'S2 905 Row 91 Spare Message German' | French: 'S2 905 Row 91 Spare Message French'
  906 = 'S2 906 Row 91 Spare Message Default' | German: 'S2 906 Row 91 Spare Message German' | French: 'S2 906 Row 91 Spare Message French'
  907 = 'S2 907 Row 91 Spare Message Default' | German: 'S2 907 Row 91 Spare Message German' | French: 'S2 907 Row 91 Spare Message French'
  908 = 'S2 908 Row 91 Spare Message Default' | German: 'S2 908 Row 91 Spare Message German' | French: 'S2 908 Row 91 Spare Message French'
  909 = 'S2 909 Row 91 Spare Message Default' | German: 'S2 909 Row 91 Spare Message German' | French: 'S2 909 Row 91 Spare Message French'
  910 = 'S2 910 Row 92 Failed To Advance.. Check Qxxx.x Default' | German: 'S2 910 Row 92 Failed To Advance.. Check Qxxx.x German' | French: 'S2 910 Row 92 Failed To Advance.. Check Qxxx.x French'
  911 = 'S2 911 Row 92 Failed To Return.. Check Qxxx.x Default' | German: 'S2 911 Row 92 Failed To Return.. Check Qxxx.x German' | French: 'S2 911 Row 92 Failed To Return.. Check Qxxx.x French'
  912 = 'S2 912 Row 92 Lost Advance Position... Check Ixxx.x Default' | German: 'S2 912 Row 92 Lost Advance Position... Check Ixxx.x German' | French: 'S2 912 Row 92 Lost Advance Position... Check Ixxx.x French'
  913 = 'S2 913 Row 92 Lost Return Position... Check Ixxx.x Default' | German: 'S2 913 Row 92 Lost Return Position... Check Ixxx.x German' | French: 'S2 913 Row 92 Lost Return Position... Check Ixxx.x French'
  914 = 'S2 914 Row 92 Switch Fault... Check Ixxx.x / Ixxx.x Default' | German: 'S2 914 Row 92 Switch Fault... Check Ixxx.x / Ixxx.x German' | French: 'S2 914 Row 92 Switch Fault... Check Ixxx.x / Ixxx.x French'
  915 = 'S2 915 Row 92 Spare Message Default' | German: 'S2 915 Row 92 Spare Message German' | French: 'S2 915 Row 92 Spare Message French'
  916 = 'S2 916 Row 92 Spare Message Default' | German: 'S2 916 Row 92 Spare Message German' | French: 'S2 916 Row 92 Spare Message French'
  917 = 'S2 917 Row 92 Spare Message Default' | German: 'S2 917 Row 92 Spare Message German' | French: 'S2 917 Row 92 Spare Message French'
  918 = 'S2 918 Row 92 Spare Message Default' | German: 'S2 918 Row 92 Spare Message German' | French: 'S2 918 Row 92 Spare Message French'
  919 = 'S2 919 Row 92 Spare Message Default' | German: 'S2 919 Row 92 Spare Message German' | French: 'S2 919 Row 92 Spare Message French'
  920 = 'S2 920 Row 93 Failed To Advance.. Check Qxxx.x Default' | German: 'S2 920 Row 93 Failed To Advance.. Check Qxxx.x German' | French: 'S2 920 Row 93 Failed To Advance.. Check Qxxx.x French'
  921 = 'S2 921 Row 93 Failed To Return.. Check Qxxx.x Default' | German: 'S2 921 Row 93 Failed To Return.. Check Qxxx.x German' | French: 'S2 921 Row 93 Failed To Return.. Check Qxxx.x French'
  922 = 'S2 922 Row 93 Lost Advance Position... Check Ixxx.x Default' | German: 'S2 922 Row 93 Lost Advance Position... Check Ixxx.x German' | French: 'S2 922 Row 93 Lost Advance Position... Check Ixxx.x French'
  923 = 'S2 923 Row 93 Lost Return Position... Check Ixxx.x Default' | German: 'S2 923 Row 93 Lost Return Position... Check Ixxx.x German' | French: 'S2 923 Row 93 Lost Return Position... Check Ixxx.x French'
  924 = 'S2 924 Row 93 Switch Fault... Check Ixxx.x / Ixxx.x Default' | German: 'S2 924 Row 93 Switch Fault... Check Ixxx.x / Ixxx.x German' | French: 'S2 924 Row 93 Switch Fault... Check Ixxx.x / Ixxx.x French'
  925 = 'S2 925 Row 93 Spare Message Default' | German: 'S2 925 Row 93 Spare Message German' | French: 'S2 925 Row 93 Spare Message French'
  926 = 'S2 926 Row 93 Spare Message Default' | German: 'S2 926 Row 93 Spare Message German' | French: 'S2 926 Row 93 Spare Message French'
  927 = 'S2 927 Row 93 Spare Message Default' | German: 'S2 927 Row 93 Spare Message German' | French: 'S2 927 Row 93 Spare Message French'
  928 = 'S2 928 Row 93 Spare Message Default' | German: 'S2 928 Row 93 Spare Message German' | French: 'S2 928 Row 93 Spare Message French'
  929 = 'S2 929 Row 93 Spare Message Default' | German: 'S2 929 Row 93 Spare Message German' | French: 'S2 929 Row 93 Spare Message French'
  930 = 'S2 930 Row 94 Failed To Advance.. Check Qxxx.x Default' | German: 'S2 930 Row 94 Failed To Advance.. Check Qxxx.x German' | French: 'S2 930 Row 94 Failed To Advance.. Check Qxxx.x French'
  931 = 'S2 931 Row 94 Failed To Return.. Check Qxxx.x Default' | German: 'S2 931 Row 94 Failed To Return.. Check Qxxx.x German' | French: 'S2 931 Row 94 Failed To Return.. Check Qxxx.x French'
  932 = 'S2 932 Row 94 Lost Advance Position... Check Ixxx.x Default' | German: 'S2 932 Row 94 Lost Advance Position... Check Ixxx.x German' | French: 'S2 932 Row 94 Lost Advance Position... Check Ixxx.x French'
  933 = 'S2 933 Row 94 Lost Return Position... Check Ixxx.x Default' | German: 'S2 933 Row 94 Lost Return Position... Check Ixxx.x German' | French: 'S2 933 Row 94 Lost Return Position... Check Ixxx.x French'
  934 = 'S2 934 Row 94 Switch Fault... Check Ixxx.x / Ixxx.x Default' | German: 'S2 934 Row 94 Switch Fault... Check Ixxx.x / Ixxx.x German' | French: 'S2 934 Row 94 Switch Fault... Check Ixxx.x / Ixxx.x French'
  935 = 'S2 935 Row 94 Spare Message Default' | German: 'S2 935 Row 94 Spare Message German' | French: 'S2 935 Row 94 Spare Message French'
  936 = 'S2 936 Row 94 Spare Message Default' | German: 'S2 936 Row 94 Spare Message German' | French: 'S2 936 Row 94 Spare Message French'
  937 = 'S2 937 Row 94 Spare Message Default' | German: 'S2 937 Row 94 Spare Message German' | French: 'S2 937 Row 94 Spare Message French'
  938 = 'S2 938 Row 94 Spare Message Default' | German: 'S2 938 Row 94 Spare Message German' | French: 'S2 938 Row 94 Spare Message French'
  939 = 'S2 939 Row 94 Spare Message Default' | German: 'S2 939 Row 94 Spare Message German' | French: 'S2 939 Row 94 Spare Message French'
  940 = 'S2 940 Row 95 Failed To Advance.. Check Qxxx.x Default' | German: 'S2 940 Row 95 Failed To Advance.. Check Qxxx.x German' | French: 'S2 940 Row 95 Failed To Advance.. Check Qxxx.x French'
  941 = 'S2 941 Row 95 Failed To Return.. Check Qxxx.x Default' | German: 'S2 941 Row 95 Failed To Return.. Check Qxxx.x German' | French: 'S2 941 Row 95 Failed To Return.. Check Qxxx.x French'
  942 = 'S2 942 Row 95 Lost Advance Position... Check Ixxx.x Default' | German: 'S2 942 Row 95 Lost Advance Position... Check Ixxx.x German' | French: 'S2 942 Row 95 Lost Advance Position... Check Ixxx.x French'
  943 = 'S2 943 Row 95 Lost Return Position... Check Ixxx.x Default' | German: 'S2 943 Row 95 Lost Return Position... Check Ixxx.x German' | French: 'S2 943 Row 95 Lost Return Position... Check Ixxx.x French'
  944 = 'S2 944 Row 95 Switch Fault... Check Ixxx.x / Ixxx.x Default' | German: 'S2 944 Row 95 Switch Fault... Check Ixxx.x / Ixxx.x German' | French: 'S2 944 Row 95 Switch Fault... Check Ixxx.x / Ixxx.x French'
  945 = 'S2 945 Row 95 Spare Message Default' | German: 'S2 945 Row 95 Spare Message German' | French: 'S2 945 Row 95 Spare Message French'
  946 = 'S2 946 Row 95 Spare Message Default' | German: 'S2 946 Row 95 Spare Message German' | French: 'S2 946 Row 95 Spare Message French'
  947 = 'S2 947 Row 95 Spare Message Default' | German: 'S2 947 Row 95 Spare Message German' | French: 'S2 947 Row 95 Spare Message French'
  948 = 'S2 948 Row 95 Spare Message Default' | German: 'S2 948 Row 95 Spare Message German' | French: 'S2 948 Row 95 Spare Message French'
  949 = 'S2 949 Row 95 Spare Message Default' | German: 'S2 949 Row 95 Spare Message German' | French: 'S2 949 Row 95 Spare Message French'
  950 = 'S2 950 Row 96 Failed To Advance.. Check Qxxx.x Default' | German: 'S2 950 Row 96 Failed To Advance.. Check Qxxx.x German' | French: 'S2 950 Row 96 Failed To Advance.. Check Qxxx.x French'
  951 = 'S2 951 Row 96 Failed To Return.. Check Qxxx.x Default' | German: 'S2 951 Row 96 Failed To Return.. Check Qxxx.x German' | French: 'S2 951 Row 96 Failed To Return.. Check Qxxx.x French'
  952 = 'S2 952 Row 96 Lost Advance Position... Check Ixxx.x Default' | German: 'S2 952 Row 96 Lost Advance Position... Check Ixxx.x German' | French: 'S2 952 Row 96 Lost Advance Position... Check Ixxx.x French'
  953 = 'S2 953 Row 96 Lost Return Position... Check Ixxx.x Default' | German: 'S2 953 Row 96 Lost Return Position... Check Ixxx.x German' | French: 'S2 953 Row 96 Lost Return Position... Check Ixxx.x French'
  954 = 'S2 954 Row 96 Switch Fault... Check Ixxx.x / Ixxx.x Default' | German: 'S2 954 Row 96 Switch Fault... Check Ixxx.x / Ixxx.x German' | French: 'S2 954 Row 96 Switch Fault... Check Ixxx.x / Ixxx.x French'
  955 = 'S2 955 Row 96 Spare Message Default' | German: 'S2 955 Row 96 Spare Message German' | French: 'S2 955 Row 96 Spare Message French'
  956 = 'S2 956 Row 96 Spare Message Default' | German: 'S2 956 Row 96 Spare Message German' | French: 'S2 956 Row 96 Spare Message French'
  957 = 'S2 957 Row 96 Spare Message Default' | German: 'S2 957 Row 96 Spare Message German' | French: 'S2 957 Row 96 Spare Message French'
  958 = 'S2 958 Row 96 Spare Message Default' | German: 'S2 958 Row 96 Spare Message German' | French: 'S2 958 Row 96 Spare Message French'
  959 = 'S2 959 Row 96 Spare Message Default' | German: 'S2 959 Row 96 Spare Message German' | French: 'S2 959 Row 96 Spare Message French'
  960 = 'S2 960 Row 97 Failed To Advance.. Check Qxxx.x Default' | German: 'S2 960 Row 97 Failed To Advance.. Check Qxxx.x German' | French: 'S2 960 Row 97 Failed To Advance.. Check Qxxx.x French'
  961 = 'S2 961 Row 97 Failed To Return.. Check Qxxx.x Default' | German: 'S2 961 Row 97 Failed To Return.. Check Qxxx.x German' | French: 'S2 961 Row 97 Failed To Return.. Check Qxxx.x French'
  962 = 'S2 962 Row 97 Lost Advance Position... Check Ixxx.x Default' | German: 'S2 962 Row 97 Lost Advance Position... Check Ixxx.x German' | French: 'S2 962 Row 97 Lost Advance Position... Check Ixxx.x French'
  963 = 'S2 963 Row 97 Lost Return Position... Check Ixxx.x Default' | German: 'S2 963 Row 97 Lost Return Position... Check Ixxx.x German' | French: 'S2 963 Row 97 Lost Return Position... Check Ixxx.x French'
  964 = 'S2 964 Row 97 Switch Fault... Check Ixxx.x / Ixxx.x Default' | German: 'S2 964 Row 97 Switch Fault... Check Ixxx.x / Ixxx.x German' | French: 'S2 964 Row 97 Switch Fault... Check Ixxx.x / Ixxx.x French'
  965 = 'S2 965 Row 97 Spare Message Default' | German: 'S2 965 Row 97 Spare Message German' | French: 'S2 965 Row 97 Spare Message French'
  966 = 'S2 966 Row 97 Spare Message Default' | German: 'S2 966 Row 97 Spare Message German' | French: 'S2 966 Row 97 Spare Message French'
  967 = 'S2 967 Row 97 Spare Message Default' | German: 'S2 967 Row 97 Spare Message German' | French: 'S2 967 Row 97 Spare Message French'
  968 = 'S2 968 Row 97 Spare Message Default' | German: 'S2 968 Row 97 Spare Message German' | French: 'S2 968 Row 97 Spare Message French'
  969 = 'S2 969 Row 97 Spare Message Default' | German: 'S2 969 Row 97 Spare Message German' | French: 'S2 969 Row 97 Spare Message French'
  970 = 'S2 970 Row 98 Failed To Advance.. Check Qxxx.x Default' | German: 'S2 970 Row 98 Failed To Advance.. Check Qxxx.x German' | French: 'S2 970 Row 98 Failed To Advance.. Check Qxxx.x French'
  971 = 'S2 971 Row 98 Failed To Return.. Check Qxxx.x Default' | German: 'S2 971 Row 98 Failed To Return.. Check Qxxx.x German' | French: 'S2 971 Row 98 Failed To Return.. Check Qxxx.x French'
  972 = 'S2 972 Row 98 Lost Advance Position... Check Ixxx.x Default' | German: 'S2 972 Row 98 Lost Advance Position... Check Ixxx.x German' | French: 'S2 972 Row 98 Lost Advance Position... Check Ixxx.x French'
  973 = 'S2 973 Row 98 Lost Return Position... Check Ixxx.x Default' | German: 'S2 973 Row 98 Lost Return Position... Check Ixxx.x German' | French: 'S2 973 Row 98 Lost Return Position... Check Ixxx.x French'
  974 = 'S2 974 Row 98 Switch Fault... Check Ixxx.x / Ixxx.x Default' | German: 'S2 974 Row 98 Switch Fault... Check Ixxx.x / Ixxx.x German' | French: 'S2 974 Row 98 Switch Fault... Check Ixxx.x / Ixxx.x French'
  975 = 'S2 975 Row 98 Spare Message Default' | German: 'S2 975 Row 98 Spare Message German' | French: 'S2 975 Row 98 Spare Message French'
  976 = 'S2 976 Row 98 Spare Message Default' | German: 'S2 976 Row 98 Spare Message German' | French: 'S2 976 Row 98 Spare Message French'
  977 = 'S2 977 Row 98 Spare Message Default' | German: 'S2 977 Row 98 Spare Message German' | French: 'S2 977 Row 98 Spare Message French'
  978 = 'S2 978 Row 98 Spare Message Default' | German: 'S2 978 Row 98 Spare Message German' | French: 'S2 978 Row 98 Spare Message French'
  979 = 'S2 979 Row 98 Spare Message Default' | German: 'S2 979 Row 98 Spare Message German' | French: 'S2 979 Row 98 Spare Message French'
  980 = 'S2 980 Row 99 Failed To Advance.. Check Qxxx.x Default' | German: 'S2 980 Row 99 Failed To Advance.. Check Qxxx.x German' | French: 'S2 980 Row 99 Failed To Advance.. Check Qxxx.x French'
  981 = 'S2 981 Row 99 Failed To Return.. Check Qxxx.x Default' | German: 'S2 981 Row 99 Failed To Return.. Check Qxxx.x German' | French: 'S2 981 Row 99 Failed To Return.. Check Qxxx.x French'
  982 = 'S2 982 Row 99 Lost Advance Position... Check Ixxx.x Default' | German: 'S2 982 Row 99 Lost Advance Position... Check Ixxx.x German' | French: 'S2 982 Row 99 Lost Advance Position... Check Ixxx.x French'
  983 = 'S2 983 Row 99 Lost Return Position... Check Ixxx.x Default' | German: 'S2 983 Row 99 Lost Return Position... Check Ixxx.x German' | French: 'S2 983 Row 99 Lost Return Position... Check Ixxx.x French'
  984 = 'S2 984 Row 99 Switch Fault... Check Ixxx.x / Ixxx.x Default' | German: 'S2 984 Row 99 Switch Fault... Check Ixxx.x / Ixxx.x German' | French: 'S2 984 Row 99 Switch Fault... Check Ixxx.x / Ixxx.x French'
  985 = 'S2 985 Row 99 Spare Message Default' | German: 'S2 985 Row 99 Spare Message German' | French: 'S2 985 Row 99 Spare Message French'
  986 = 'S2 986 Row 99 Spare Message Default' | German: 'S2 986 Row 99 Spare Message German' | French: 'S2 986 Row 99 Spare Message French'
  987 = 'S2 987 Row 99 Spare Message Default' | German: 'S2 987 Row 99 Spare Message German' | French: 'S2 987 Row 99 Spare Message French'
  988 = 'S2 988 Row 99 Spare Message Default' | German: 'S2 988 Row 99 Spare Message German' | French: 'S2 988 Row 99 Spare Message French'
  989 = 'S2 989 Row 99 Spare Message Default' | German: 'S2 989 Row 99 Spare Message German' | French: 'S2 989 Row 99 Spare Message French'
  990 = 'S2 990 Row 100 Failed To Advance.. Check Qxxx.x Default' | German: 'S2 990 Row 100 Failed To Advance.. Check Qxxx.x German' | French: 'S2 990 Row 100 Failed To Advance.. Check Qxxx.x French'
  991 = 'S2 991 Row 100 Failed To Return.. Check Qxxx.x Default' | German: 'S2 991 Row 100 Failed To Return.. Check Qxxx.x German' | French: 'S2 991 Row 100 Failed To Return.. Check Qxxx.x French'
  992 = 'S2 992 Row 100 Lost Advance Position... Check Ixxx.x Default' | German: 'S2 992 Row 100 Lost Advance Position... Check Ixxx.x German' | French: 'S2 992 Row 100 Lost Advance Position... Check Ixxx.x French'
  993 = 'S2 993 Row 100 Lost Return Position... Check Ixxx.x Default' | German: 'S2 993 Row 100 Lost Return Position... Check Ixxx.x German' | French: 'S2 993 Row 100 Lost Return Position... Check Ixxx.x French'
  994 = 'S2 994 Row 100 Switch Fault... Check Ixxx.x / Ixxx.x Default' | German: 'S2 994 Row 100 Switch Fault... Check Ixxx.x / Ixxx.x German' | French: 'S2 994 Row 100 Switch Fault... Check Ixxx.x / Ixxx.x French'
  995 = 'S2 995 Row 100 Spare Message Default' | German: 'S2 995 Row 100 Spare Message German' | French: 'S2 995 Row 100 Spare Message French'
  996 = 'S2 996 Row 100 Spare Message Default' | German: 'S2 996 Row 100 Spare Message German' | French: 'S2 996 Row 100 Spare Message French'
  997 = 'S2 997 Row 100 Spare Message Default' | German: 'S2 997 Row 100 Spare Message German' | French: 'S2 997 Row 100 Spare Message French'
  998 = 'S2 998 Row 100 Spare Message Default' | German: 'S2 998 Row 100 Spare Message German' | French: 'S2 998 Row 100 Spare Message French'
  999 = 'S2 999 Row 100 Spare Message Default' | German: 'S2 999 Row 100 Spare Message German' | French: 'S2 999 Row 100 Spare Message French'
  1000 = 'S2_Alarms Default 1000' | German: 'S2_Alarms German 1000' | French: 'S2_Alarms French 1000'
   = ''
END_TEXTLIST

(* stored: Version 1.1.0.1, ProductVersion 3.1.4024.12
   TextList S2_Alarms: Id {7e858b91-f198-414f-b5ed-956d732631aa} *)
